// TIA Portal project "3 Tane Pozitif KT ile Basma Sayan Uygulaması" (V18)

(* hardware
DEVICE "S7-1200 station_1"  S7-1200 Station
   slot 0: "Rack_0"  S7-1200 Rack  Rack  V1.0
   slot 1: "PLC_1"  CPU 1214C AC/DC/Rly  6ES7 214-1BG40-0XB0  V4.6
*)

// ===== PLC "PLC_1"  CPU 1214C AC/DC/Rly =====

VAR_GLOBAL   // PLC tag table "Default tag table"
   "Stop" AT %I0.0 : Bool;
   "PKT_1" AT %I0.1 : Bool;
   "PKT_2" AT %I0.2 : Bool;
   "PKT_Yardımcı_1" AT %M0.0 : Bool;
   "Motor_1" AT %Q0.0 : Bool;
   "PKT_Yardımcı_2" AT %M0.1 : Bool;
   "PKT_3" AT %I0.3 : Bool;
   "PKT_Yardımcı_3" AT %M0.2 : Bool;
END_VAR

ORGANIZATION_BLOCK "Main"   // OB1, LAD, ProgramCycle
TITLE = "Main Program Sweep (Cycle)"
{ S7_Optimized_Access := 'TRUE' }
VERSION : 0.1
// ÜÇ AYRI YERDEN TEK BUTONLA START STOP
   VAR_INPUT
      Initial_Call : Bool;   // Initial call of this OB
      Remanence : Bool;   // =True, if remanent data are available
   END_VAR
   VAR_TEMP   // added for the SCL form of the ladder/FBD networks
      _w1 : Bool;
      _w2 : Bool;
      _w3 : Bool;
      _w4 : Bool;
   END_VAR
BEGIN

REGION Network 1
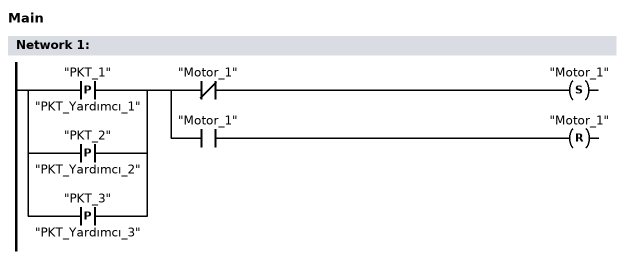
   RUNG wire#powerrail
      P_Contact(operand := "PKT_1", bit := "PKT_Yardımcı_1")
      wire#w1
      I_Contact( "Motor_1" )
      S_Coil( "Motor_1" )
   END_RUNG
   RUNG wire#powerrail
      P_Contact(operand := "PKT_2", bit := "PKT_Yardımcı_2")
   END_RUNG wire#w1
   RUNG wire#powerrail
      P_Contact(operand := "PKT_3", bit := "PKT_Yardımcı_3")
   END_RUNG wire#w1
   RUNG wire#w1
      Contact( "Motor_1" )
      R_Coil( "Motor_1" )
   END_RUNG
   // the same network as SCL:
   #_w1 := "PKT_1" AND NOT "PKT_Yardımcı_1";   // rising edge of "PKT_1"
   "PKT_Yardımcı_1" := "PKT_1";
   #_w2 := "PKT_2" AND NOT "PKT_Yardımcı_2";   // rising edge of "PKT_2"
   "PKT_Yardımcı_2" := "PKT_2";
   #_w3 := "PKT_3" AND NOT "PKT_Yardımcı_3";   // rising edge of "PKT_3"
   "PKT_Yardımcı_3" := "PKT_3";
   #_w4 := #_w1 OR #_w2 OR #_w3;
   IF #_w4 AND NOT "Motor_1" THEN "Motor_1" := TRUE; END_IF;
   IF #_w4 AND "Motor_1" THEN "Motor_1" := FALSE; END_IF;
END_REGION
END_ORGANIZATION_BLOCK